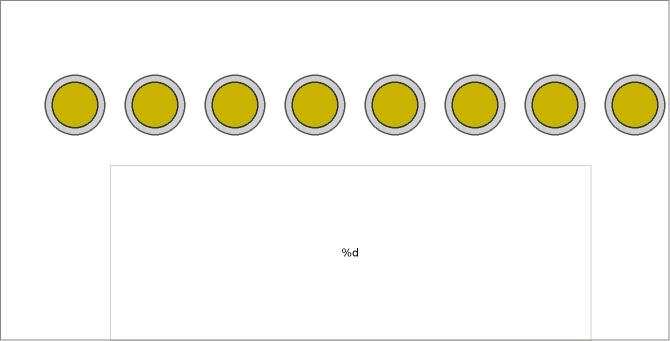
VISUALIZATION byteCounter  // 670x341
    Lamp1 (120,70 70x70), variable: byteCounter.bitRep[6], style: Lamp-Lamp1-Yellow
    Lamp1 (40,70 70x70), variable: byteCounter.bitRep[7], style: Lamp-Lamp1-Yellow
    Lamp1 (280,70 70x70), variable: byteCounter.bitRep[4], style: Lamp-Lamp1-Yellow
    Lamp1 (200,70 70x70), variable: byteCounter.bitRep[5], style: Lamp-Lamp1-Yellow
    Lamp1 (440,70 70x70), variable: byteCounter.bitRep[2], style: Lamp-Lamp1-Yellow
    Lamp1 (360,70 70x70), variable: byteCounter.bitRep[3], style: Lamp-Lamp1-Yellow
    Lamp1 (600,70 70x70), variable: byteCounter.bitRep[0], style: Lamp-Lamp1-Yellow
    Lamp1 (520,70 70x70), variable: byteCounter.bitRep[1], style: Lamp-Lamp1-Yellow
    Textfield (110,165 481x176), "%d", text variable: byteCounter.byteCount
END_VISUALIZATION

(* stored: Version 1.1.0.1, ProductVersion 3.1.4024.5
   Visu byteCounter: Id {daba41cc-d7c7-4c60-b753-d9093596e15e} *)
